Staubli VAL3: EDITNUM.pgx

public program editNum(string& x_sItem, string& x_sItemValue, num& x_nValue, num x_nSelect)
  local string l_sEmpty
  local num l_nValue
  local bool l_bRes
  local num l_nKey
  local num l_nPos
begin
  //
  do
    call clear(0,13)
    call findPos(x_sItem,":",l_nPos)
    gotoxy(nTopX+1,nTopY+nView+1)
    setTextMode(0)
    put(x_sItem)
    call strlength(l_sEmpty,nBottomX-l_nPos+1)
    call type(nTopX+l_nPos+2,nTopY+nView+1,l_sEmpty)
    gotoxy(nTopX+l_nPos+2,nTopY+nView+1)
    toNum(x_sItemValue,l_nValue,l_bRes)
    l_nKey=get(l_nValue)
    if l_nKey==270
      x_sItemValue=toString(".3",l_nValue)
      x_nValue=l_nValue
    endIf
    call strfill(x_sItem,l_nPos+1,x_sItem)
    x_sItem=x_sItem+x_sItemValue
    call strlength(x_sItem,nBottomX+1)
    gotoxy(nTopX+1,nTopY+nView+1)
    setTextMode(1)
    call type(nTopX+1,nTopY+nView+1,x_sItem)
    setTextMode(0)
    delay(0)
  until l_nKey==270 or l_nKey==255

end
